# EPICS StreamDevice protocol: helloWorldIOCApp/Db/arduino.proto
Terminator = LF;
get_analog {
    out "R";
    in "R %f";
    ExtraInput = Ignore;
}
set_digital {
    out "W%d\n";
    ExtraInput = Ignore;
}
